FUNCTION_BLOCK fbStep
VAR_INPUT
	/// // previous step completed 
	xPreviousStepComplete: BOOL;
	/// Step should stay active until this flag is set TRUE 
	xStepDone: BOOL;
END_VAR
VAR_OUTPUT
	/// Until external logic signals "done", this step status is FALSE, if the external logic signals done, this step is completed 
	xStepComplete: BOOL;
	/// This flag should be used to steer a codition 
	xStepInProgress: BOOL;
END_VAR

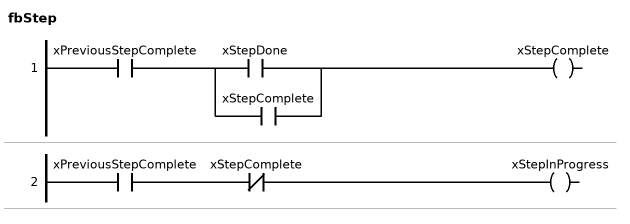
// NETWORK 1
xStepComplete := xPreviousStepComplete AND (xStepDone OR xStepComplete);

// NETWORK 2
xStepInProgress := xPreviousStepComplete AND NOT xStepComplete;

END_FUNCTION_BLOCK

(* stored: Version 1.1.0.1, ProductVersion 3.1.4024.12
   POU fbStep: Id {36f01f99-9b95-4679-bf75-e74beaa38c02}, SpecialFunc None *)
